FUNCTION FUN_GetHighByte : BYTE
VAR_INPUT
	wIn			:WORD;			
END_VAR
VAR
	byHigh		:BYTE;
END_VAR


// Get the high byte value from the word
byHigh.0 := wIn.8;
byHigh.1 := wIn.9;
byHigh.2 := wIn.10;
byHigh.3 := wIn.11;
byHigh.4 := wIn.12;
byHigh.5 := wIn.13;
byHigh.6 := wIn.14;
byHigh.7 := wIn.15;

// Return value
FUN_GetHighByte := byHigh;

END_FUNCTION

(* stored: Version 1.1.0.1, ProductVersion 3.1.4024.12
   POU FUN_GetHighByte: Id {67e627d9-9694-492f-8813-a4d6fd056bfe}, SpecialFunc None *)
